INTERFACE I_AxisGear EXTENDS I_Base

METHOD GearIn
VAR_INPUT
END_VAR
END_METHOD

PROPERTY GearInMultiMasterOptions : ST_GearInMultiMasterOptions
SET
END_SET
END_PROPERTY

METHOD GearOut
VAR_INPUT
END_VAR
END_METHOD

{attribute 'monitoring' := 'call'}
PROPERTY GearRatioMaster1 : LREAL
SET
END_SET
END_PROPERTY

{attribute 'monitoring' := 'call'}
PROPERTY GearRatioMaster2 : LREAL
SET
END_SET
END_PROPERTY

{attribute 'monitoring' := 'call'}
PROPERTY GearRatioMaster3 : LREAL
SET
END_SET
END_PROPERTY

{attribute 'monitoring' := 'call'}
PROPERTY GearRatioMaster4 : LREAL
SET
END_SET
END_PROPERTY

PROPERTY Master1 : I_Axis
SET
END_SET
END_PROPERTY

PROPERTY Master2 : I_Axis
SET
END_SET
END_PROPERTY

PROPERTY Master3 : I_Axis
SET
END_SET
END_PROPERTY

PROPERTY Master4 : I_Axis
SET
END_SET
END_PROPERTY

END_INTERFACE

(* stored: Version 1.1.0.1, ProductVersion 3.1.4026.18
   Itf I_AxisGear: Id {6c275f38-a60b-4115-a407-e89a6c7e3629}
   Method GearIn: Id {38ea9e4e-cf72-4cc7-8c20-73160004533f}
   Property GearInMultiMasterOptions: Id {613feb86-6752-4536-9fc8-bfe1bdab419f}
   Set Set: Id {e5da6742-8725-45eb-9b70-46c8b0ab084b}
   Method GearOut: Id {815649dc-88ad-44e1-a7a8-4b99a60da25c}
   Property GearRatioMaster1: Id {4b5bfddc-e3c1-4e0d-a62a-4ac1c748af24}
   Set Set: Id {7985490c-9483-4e53-840b-60d0214e5d5b}
   Property GearRatioMaster2: Id {9c73a257-c796-4dc4-9448-01ff526cdfbb}
   Set Set: Id {c4d6ae08-cdcd-4e30-9a0f-e5358ec8852d}
   Property GearRatioMaster3: Id {7c9271b0-ed38-4604-ba81-d8378bbd6503}
   Set Set: Id {b4955f86-4638-4c42-b841-bf8f5f197ea4}
   Property GearRatioMaster4: Id {a047fd92-9041-4d61-91a8-746935a1f243}
   Set Set: Id {0e681c72-6e98-4841-901c-9219d55c1efe}
   Property Master1: Id {843a1922-1c9e-4cfe-bfc1-1ac03b6b18ae}
   Set Set: Id {f5ac2ce0-2c01-4041-83c2-c67e4a02ae09}
   Property Master2: Id {cd1a16a8-2ae3-41bd-88ba-fb6123180948}
   Set Set: Id {43b7fa19-ad7f-4316-b2c3-ca00e459f34a}
   Property Master3: Id {628628f6-c99d-4907-9b3f-945f9c7b9f75}
   Set Set: Id {867c7ce7-40a8-4e21-a4a1-642bf6c643ab}
   Property Master4: Id {61c1edd3-cd5b-4fc2-8356-3ed01c07d3dd}
   Set Set: Id {31b5d25f-e1fb-42c1-b9c8-b368e3a69491} *)
